INTERFACE IStation

METHOD Abort : BOOL
VAR_INPUT
END_VAR
END_METHOD

METHOD HasMover : BOOL
VAR_INPUT
	mover : IMover;
END_VAR
END_METHOD

METHOD IsClear : BOOL
VAR_INPUT
END_VAR
END_METHOD

METHOD isComplete : BOOL
VAR_INPUT
END_VAR
END_METHOD

PROPERTY IsLastStation : BOOL
GET
END_GET
SET
END_SET
END_PROPERTY

METHOD IsOperating : BOOL
VAR_INPUT
END_VAR
END_METHOD

METHOD IsReady : BOOL
VAR_INPUT
END_VAR
END_METHOD

METHOD MoverAway : BOOL
VAR_INPUT
END_VAR
END_METHOD

PROPERTY Position : MC_LREAL
GET
END_GET
SET
END_SET
END_PROPERTY

END_INTERFACE

(* stored: Version 1.1.0.1, ProductVersion 3.1.4024.12
   Itf IStation: Id {485e049e-0dbf-4cb2-92d5-eeadda868244}
   Method Abort: Id {b28dc0f6-87fc-48d7-a2b8-a7b3817f6bfc}
   Method HasMover: Id {899154dd-dc96-481c-8916-04ef12eb0809}
   Method IsClear: Id {dac8382a-5be0-4583-b95c-60e24b8b6b4e}
   Method isComplete: Id {f04ef912-a2d5-4671-bb7a-85761f45eebd}
   Property IsLastStation: Id {53217bec-eab6-4401-b1af-a6e405784e44}
   Get Get: Id {16b9a74e-183d-4495-8d6b-7aad46c030c0}
   Set Set: Id {0aad8e63-8a10-47b1-88ed-3a7470833511}
   Method IsOperating: Id {e194a704-bfb6-44e5-ad98-14da5789c4a2}
   Method IsReady: Id {dc79e32c-78a1-4756-8757-7f3281e1b29e}
   Method MoverAway: Id {fe173456-b154-4b4b-8d80-d2a0e72f7087}
   Property Position: Id {9ae5a97b-2f21-4be5-9e8a-7a6419e2618c}
   Get Get: Id {4a419836-b78e-4e9e-986b-a3127f385808}
   Set Set: Id {c0a16b0f-042c-4777-afba-11949a5791fc} *)
